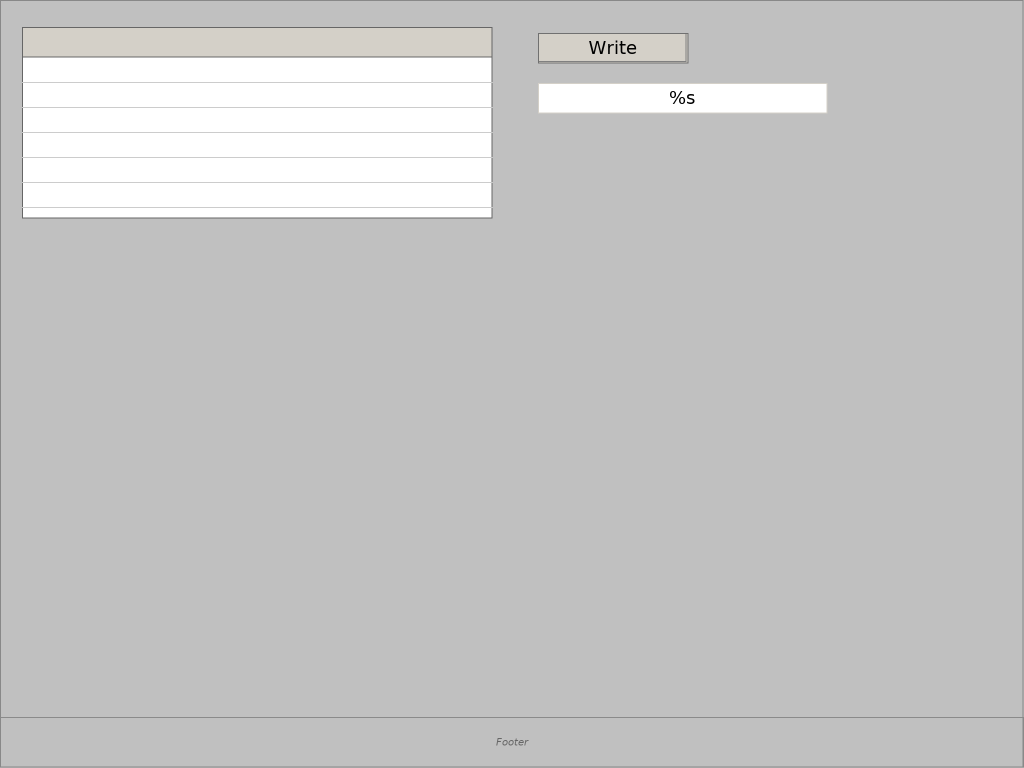
VISUALIZATION Writing  // 1024x768
    Table (22,27 470x191), data array: GVL.data
        p3854506369: GVL.data[INDEX].field01
        p1892666644: GVL.data[INDEX].field02
        p338671338: GVL.data[INDEX].field03
        p2170511999: GVL.data[INDEX].field04
        p3723444502: GVL.data[INDEX].field05
        p2232123230: Field 01
        p511219082: Field 02
        p1755163831: Field 03
        p4092479075: Field 04
        p2237128397: Field 05
    Button (538,33 150x30), "Write"
        tap GVL.recordFileNow
    Textfield (538,83 289x30), "%s", text variable: GVL.sFileName
        OnMouseClick: write the text variable via Default
    Frame (0,717 1024x50)
        shows Footer()
END_VISUALIZATION

(* stored: Version 1.1.0.1, ProductVersion 3.1.4024.13
   Visu Writing: Id {92d123c7-81c9-4e56-b29d-edea5cefc885} *)
